FUNCTION_BLOCK StationFactory EXTENDS Factory
VAR
	prtStation : POINTER TO Station;
	itfStation : ITF_Station;
END_VAR

METHOD Create : ITF_Cyclic
VAR_INPUT
END_VAR
prtStation := __NEW(Station);
Create := prtStation^;
IF __QUERYINTERFACE(Create,itfStation) THEN
	itfStation.Position := 1250.0;
END_IF
END_METHOD

END_FUNCTION_BLOCK

(* stored: Version 1.1.0.1, ProductVersion 3.1.4024.12
   POU StationFactory: Id {ec7bc97c-7694-4de4-87d3-7cdc42a01c44}, SpecialFunc None
   Method Create: Id {19cdbfb2-061f-48cf-890b-7bc2c6665293} *)
